// TwinCAT 3 PLC project AOC2016
// ProgramVersion: 3.1.4024.12
// libraries:
//   Tc2_Standard, * (Beckhoff Automation GmbH)
//   Tc2_System, * (Beckhoff Automation GmbH)
//   Tc3_Module, * (Beckhoff Automation GmbH)
//   TcUnit, * (www.tcunit.org)
// project tree:
//   MAIN/ MAIN.TcPOU
//   / PlcTask.TcTTO
//   POUs/ Common.TcPOU, Day1.TcPOU
// real-time tasks:
//   TASK PlcTask: cycle T#10ms, priority 20, ADS port 350

CONFIGURATION AOC2016
    RESOURCE PLC ON TwinCAT3
        TASK PlcTask(INTERVAL := T#10ms, PRIORITY := 20);
        PROGRAM MAIN WITH PlcTask : MAIN;
    END_RESOURCE
END_CONFIGURATION

// ---- MAIN/MAIN.TcPOU
PROGRAM MAIN
VAR
	Day1 : Day1;
END_VAR

TcUnit.RUN();

END_PROGRAM

// ---- POUs/Day1.TcPOU
FUNCTION_BLOCK Day1 EXTENDS Common
VAR
	
	
END_VAR

END_FUNCTION_BLOCK

// ---- POUs/Common.TcPOU
FUNCTION_BLOCK Common
VAR
	_sSrcNetId		: T_AmsNetId;
	_tTimeout		: TIME := DEFAULT_ADS_TIMEOUT;
END_VAR

METHOD openFile
VAR
	fileOpen : FB_FileOpen;
	sSrcNetID : T_AmsNetId := '127.0.0.1.1.1';
END_VAR
VAR_IN_OUT
	hFile : UINT;
END_VAR
VAR_INPUT
	sSrcPathName : T_MaxString;
END_VAR
VAR_INST
	stepper : DINT;
END_VAR
CASE stepper OF
0:
	fileOpen(bExecute := FALSE);
	fileOpen(sNetId := sSrcNetId, sPathName := sSrcPathName, 
                         nMode := FOPEN_MODEREAD OR FOPEN_MODEBINARY, 
                         ePath := PATH_GENERIC, tTimeout := _tTimeOut, bExecute := TRUE );
	stepper := stepper + 1;
1:
	
END_CASE
END_METHOD

END_FUNCTION_BLOCK
